// TIA Portal V18 export
// export: Created 2026-03-12T16:04:35.2244001Z, ExportSetting WithDefaults, DisplayName Totally Integrated Automation Portal, DisplayVersion V18 Update 5, DisplayName TIA Portal Openness, DisplayVersion V18 Update 5, DisplayName TIA Portal Version Control Interface, DisplayVersion V18, DisplayName SINAMICS Startdrive Advanced, DisplayVersion V18, DisplayName SINAMICS Startdrive G130, G150, S120, S150, SINAMICS MV, S210, DisplayVersion V18, DisplayName SINAMICS Startdrive G110M, G120, G120C, G120D, G120P, G115D, DisplayVersion V18, DisplayName STEP 7 Professional, DisplayVersion V18 Update 5, DisplayName STEP 7 Safety, DisplayVersion V18, DisplayName WinCC Professional, DisplayVersion V18 Update 5
FUNCTION_BLOCK "FB STATUS ECSX"   // FB12, LAD
TITLE = Function Block STATUS ECSX - Status dos exaustores (ECS1 - ECS2 - ECS3)
{ S7_Optimized_Access := 'TRUE' }
VERSION : 0.1
// Sinais de status (ligado e falha) recebidos de campo
// stored: AutoNumber false, IsIECCheckEnabled false, IsRetainMemResEnabled false, MemoryReserve 100, SetENOAutomatically false, UDAEnableTagReadback false
   VAR_INPUT
      INPUT_LIGADO : Bool;   // Entrada do sinal de Motor/Bomba ligado
      INPUT_FALHA : Bool;   // Entrada do sinal de falha instanciado na Network 1
      INPUT_MANUTEN : Bool;   // Entrada do sinal de manutenção instanciado na Network 1
      INPUT_FALHA_PROFINET : Bool;   // 1 = Indica falta de comunicação PROFINET com o equipamento
   END_VAR
   VAR_OUTPUT
      STATUS_MOTOR : Byte;   // Indicador de Status do exaustor
   END_VAR
BEGIN

REGION Network 1: Acionamento do status ligado
   // INUPT_LIGADO = TRUE: Exaustor ligado
   // INPUT_FALHA = TRUE: Exaustor em falha
   // INPUT_FALHA_PROFINET = TRUE: Sem Comunicação PROFINET
   // INPUT_MANUTEN = TRUE: Soprador/Exaustor em manutenção
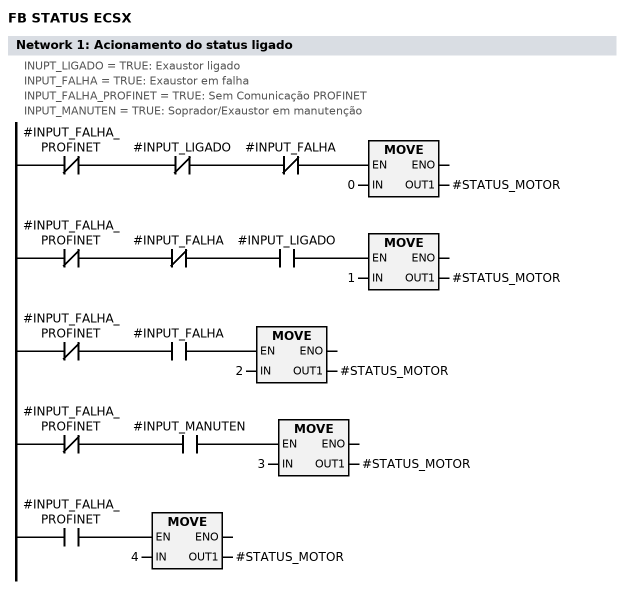
   RUNG wire#powerrail
      I_Contact( #INPUT_FALHA_PROFINET )
      I_Contact( #INPUT_LIGADO )
      I_Contact( #INPUT_FALHA )
      Move(in := 0, out1 => #STATUS_MOTOR)
   END_RUNG
   RUNG wire#powerrail
      I_Contact( #INPUT_FALHA_PROFINET )
      I_Contact( #INPUT_FALHA )
      Contact( #INPUT_LIGADO )
      Move(in := 1, out1 => #STATUS_MOTOR)
   END_RUNG
   RUNG wire#powerrail
      I_Contact( #INPUT_FALHA_PROFINET )
      Contact( #INPUT_FALHA )
      Move(in := 2, out1 => #STATUS_MOTOR)
   END_RUNG
   RUNG wire#powerrail
      I_Contact( #INPUT_FALHA_PROFINET )
      Contact( #INPUT_MANUTEN )
      Move(in := 3, out1 => #STATUS_MOTOR)
   END_RUNG
   RUNG wire#powerrail
      Contact( #INPUT_FALHA_PROFINET )
      Move(in := 4, out1 => #STATUS_MOTOR)
   END_RUNG
   // the same network as SCL:
   IF NOT #INPUT_FALHA_PROFINET AND NOT #INPUT_LIGADO AND NOT #INPUT_FALHA THEN #STATUS_MOTOR := 0; END_IF;
   IF NOT #INPUT_FALHA_PROFINET AND NOT #INPUT_FALHA AND #INPUT_LIGADO THEN #STATUS_MOTOR := 1; END_IF;
   IF NOT #INPUT_FALHA_PROFINET AND #INPUT_FALHA THEN #STATUS_MOTOR := 2; END_IF;
   IF NOT #INPUT_FALHA_PROFINET AND #INPUT_MANUTEN THEN #STATUS_MOTOR := 3; END_IF;
   IF #INPUT_FALHA_PROFINET THEN #STATUS_MOTOR := 4; END_IF;
END_REGION
END_FUNCTION_BLOCK
